	_Done : BOOL;
	_State : DB_COMMAND_EXECUTION_STATE;
	_GetError : BOOL;
	_Logger : Tc3_EventLogger.I_TcMessage;	
	_Connected : BOOL;
	_DataSetLoaded : BOOL;
	_DisconnectingState : DB_COMMAND_DISCONNECTING_STATE;
	_LastException : Exception;
END_VAR

{attribute 'monitoring' := 'call'}
{attribute 'OPC.UA.DA.Property' := '1'}
{attribute 'OPC.UA.DA.Access' := '1'}
PROPERTY Busy : BOOL
GET
Busy := State <> DB_COMMAND_EXECUTION_STATE.IDLING;
END_GET
END_PROPERTY

{attribute 'monitoring' := 'call'}
PROPERTY ClassName : REFERENCE TO STRING
GET
ClassName REF= _ClassName;
END_GET
END_PROPERTY

{attribute 'monitoring' := 'call'}
{attribute 'OPC.UA.DA.Property' := '1'}
{attribute 'OPC.UA.DA.Access' := '1'}
PROPERTY CommandText : REFERENCE TO Tc2_System.T_MaxString
GET
CommandText REF= _ExecutionParameters.CommandText;
END_GET
END_PROPERTY

{attribute 'monitoring' := 'call'}
{attribute 'OPC.UA.DA.Property' := '1'}
{attribute 'OPC.UA.DA.Access' := '1'}
PROPERTY Done : BOOL
GET
Done := _Done;
END_GET
END_PROPERTY

{attribute 'monitoring' := 'call'}
{attribute 'OPC.UA.DA.Property' := '1'}
{attribute 'OPC.UA.DA.Access' := '1'}
PROPERTY Error : BOOL
GET
Error := State = DB_COMMAND_EXECUTION_STATE.IDLING AND_THEN NOT _LastException.Empty;
END_GET
END_PROPERTY

METHOD Execute
VAR
	requestEventTextError : BOOL;	
	requestEventTextErrorCode : HRESULT;
END_VAR
VAR_INST
	errorMessage : STRING(255);	
END_VAR
START:

IF NOT _LastException.Empty THEN
	_GetError := FALSE;
END_IF

IF _GetError THEN
	IF _Logger <> 0 THEN 
		IF _Logger.RequestEventText(
			1033,
			errorMessage,
			SIZEOF(errorMessage),
			bError => requestEventTextError,
			hrErrorCode => requestEventTextErrorCode
		) THEN
			IF requestEventTextError THEN					
				errorMessage := String.Concat2('_Logger.RequestEventText() call error. Error code is ', TO_STRING(requestEventTextErrorCode));
			END_IF
		ELSE
			RETURN;
		END_IF			
	ELSE
		errorMessage :=  'Logger is not specified';
	END_IF				
	
	_LastExceptionHelper.Throw(
		0,
		TO_WSTRING(errorMessage),
		__POUNAME(),
		ClassName,
		CurrentNamespace.Name,
		__POSITION(
	)
	);
	JMP START;	
END_IF

CASE State OF
	DB_COMMAND_EXECUTION_STATE.STARTING:
		MEMSET(destAddr := _ExecutionParameters.TargetBuffer, fillByte := 0, n := _ExecutionParameters.TargetBufferSize);	
		_State := DB_COMMAND_EXECUTION_STATE.CONNECTING;		
		JMP START;		
	
	DB_COMMAND_EXECUTION_STATE.CONNECTING:
		IF _DbConnection.Connect(hDBID := _ExecutionParameters.DBID) THEN
			IF _DbConnection.bError THEN
				_GetError := TRUE;
				_Logger := _DbConnection.ipTcResult;
				_State := DB_COMMAND_EXECUTION_STATE.DISCONNECTING;				
			ELSE
				_Connected := TRUE;
				_State := DB_COMMAND_EXECUTION_STATE.PREPARING;
			END_IF
			
			JMP START;
		END_IF
	
	DB_COMMAND_EXECUTION_STATE.PREPARING:
		IF _DbConnection.CreateCmd(ADR(_Command)) THEN
			IF _DbConnection.bError THEN
				_GetError := TRUE;
				_Logger := _DbConnection.ipTcResult;
				_State := DB_COMMAND_EXECUTION_STATE.DISCONNECTING;				
			ELSE
				_State := DB_COMMAND_EXECUTION_STATE.EXECUTING;
			END_IF
			
			JMP START;
		END_IF
	
	DB_COMMAND_EXECUTION_STATE.EXECUTING:
		IF _ExecutionParameters.MaxRecordsToReadAtTime = 0 THEN
			IF _Command.Execute(ADR(_ExecutionParameters.CommandText), SIZEOF(_ExecutionParameters.CommandText)) THEN
				IF _Command.bError THEN
					_GetError := TRUE;
					_Logger := _Command.ipTcResult;
				END_IF
				
				_State := DB_COMMAND_EXECUTION_STATE.DISCONNECTING;
				
				JMP START;			
			END_IF
		ELSE
			IF _Command.ExecuteDataReturn(ADR(_ExecutionParameters.CommandText), SIZEOF(_ExecutionParameters.CommandText), ADR(_SQLResult)) THEN
				IF _Command.bError THEN
					_GetError := TRUE;
					_Logger := _Command.ipTcResult;
					_State := DB_COMMAND_EXECUTION_STATE.DISCONNECTING;
				ELSE
					_State := DB_COMMAND_EXECUTION_STATE.LOADING_RESULT_DATA_SET;
				END_IF
				
				JMP START;			
			END_IF
		END_IF
		
	DB_COMMAND_EXECUTION_STATE.LOADING_RESULT_DATA_SET:
		IF _SQLResult.Read(
			0,
			_ExecutionParameters.MaxRecordsToReadAtTime,
			_ExecutionParameters.TargetBuffer,
			_ExecutionParameters.TargetBufferSize,
			TRUE,
			TRUE
		) THEN
			IF _SQLResult.bError THEN
				_GetError := TRUE;
				_SQLResult.Release();
				_Logger := _SQLResult.ipTcResult;
			ELSE
				_DataSetLoaded := TRUE;
			END_IF

			_State := DB_COMMAND_EXECUTION_STATE.DISCONNECTING;
			
			JMP START;			
		END_IF

	DB_COMMAND_EXECUTION_STATE.DISCONNECTING:
		CASE _DisconnectingState OF
			DB_COMMAND_DISCONNECTING_STATE.IDLING:
				IF _DataSetLoaded THEN
					_DisconnectingState := DB_COMMAND_DISCONNECTING_STATE.DATA_SET_RELEASING;
				ELSIF _Connected THEN
					_DisconnectingState := DB_COMMAND_DISCONNECTING_STATE.DISCONNECTING;					
				ELSE
					_State := DB_COMMAND_EXECUTION_STATE.IDLING;	
					_Done := _LastException.Empty;	
				END_IF
				
				JMP START;
				
			DB_COMMAND_DISCONNECTING_STATE.DATA_SET_RELEASING:
				IF _SQLResult.Release() THEN
					_DataSetLoaded := FALSE;
					_DisconnectingState := DB_COMMAND_DISCONNECTING_STATE.DISCONNECTING;
					JMP START;										
				END_IF
				
			DB_COMMAND_DISCONNECTING_STATE.DISCONNECTING:
				IF _DbConnection.Disconnect() THEN
					_Connected := FALSE;
					_DisconnectingState := DB_COMMAND_DISCONNECTING_STATE.IDLING;
					JMP START;										
				END_IF
		END_CASE	
END_CASE
END_METHOD

{attribute 'monitoring' := 'call'}
{attribute 'OPC.UA.DA.Property' := '1'}
{attribute 'OPC.UA.DA.Access' := '1'}
PROPERTY LastException : REFERENCE TO Exception
GET
LastException REF= _LastException;
END_GET
END_PROPERTY

METHOD Reset
VAR_OUTPUT
	exception : Exception;
END_VAR
IF Busy THEN
	_LastExceptionHelper.Throw(
		0,
		"Previous command execution is not finished",
		__POUNAME(),
		ClassName,
		CurrentNamespace.Name,
		__POSITION(
	)
	); 
	RETURN;
END_IF

_Done := FALSE;
_State := DB_COMMAND_EXECUTION_STATE.STARTING;
_GetError := FALSE;
_Logger := 0;	
_Connected := FALSE;
_DataSetLoaded := FALSE;
_DisconnectingState := DB_COMMAND_DISCONNECTING_STATE.IDLING;
_LastException.Clear();
END_METHOD

METHOD Start 
VAR_INPUT
	dbId : UDINT;
	commandText : Tc2_System.T_MaxString;
	targetBuffer : PVOID;
	targetBufferSize : UDINT;
	maxRecordsToReadAtTime : UINT;
END_VAR
VAR_OUTPUT
	exception : Exception;
END_VAR
VAR
	executionParameters : POINTER TO DB_COMMAND_EXECUTION_PARAMETERS;
END_VAR
IF Busy THEN
	_LastExceptionHelper.Throw(
		0,
		"Previous command execution is not finished",
		__POUNAME(),
		ClassName,
		CurrentNamespace.Name,
		__POSITION(
	)
	); 
	RETURN;
END_IF

IF maxRecordsToReadAtTime > 0 AND_THEN (targetBuffer = 0 OR_ELSE targetBufferSize = 0) THEN
	_LastExceptionHelper.Throw(
		0,
		"Parameter 'maxRecordsToReadAtTime' is greater then zero, but 'targetBuffer' or 'targetBufferSize' has incorrect values",
		__POUNAME(),
		ClassName,
		CurrentNamespace.Name,
		__POSITION(
	)
	);
	RETURN;
END_IF

_ExecutionParameters.DbId := dbId;
_ExecutionParameters.CommandText := commandText;
_ExecutionParameters.TargetBuffer := targetBuffer; 
_ExecutionParameters.TargetBufferSize := targetBufferSize;
_ExecutionParameters.MaxRecordsToReadAtTime := maxRecordsToReadAtTime;

Reset();
END_METHOD

{attribute 'monitoring' := 'call'}
{attribute 'OPC.UA.DA.Property' := '1'}
{attribute 'OPC.UA.DA.Access' := '1'}
PROPERTY State : DB_COMMAND_EXECUTION_STATE
GET
State := _State;
END_GET
END_PROPERTY

{attribute 'monitoring' := 'call'}
{attribute 'OPC.UA.DA.Property' := '1'}
{attribute 'OPC.UA.DA.Access' := '1'}
PROPERTY Timeout : TIME
GET
Timeout := _Command.tTimeout;
END_GET
SET
_Command.tTimeout := Timeout;
_SQLResult.tTimeout := Timeout;
END_SET
END_PROPERTY

END_FUNCTION_BLOCK

// ---- Database/StoredProcedure/DbProcedureExecutor.TcPOU
{attribute 'no_explicit_call' := 'do not call this function block directly'}
FUNCTION_BLOCK DbProcedureExecutor EXTENDS TC.ToolkitObject IMPLEMENTS TC.IAction
VAR_STAT
	//! <summary>Class name shared by all instances of this function block.</summary>
	_ClassName : STRING := __POUNAME();
END_VAR
VAR	
	_DbConnection : Tc3_Database.FB_SQLDatabaseEvt(sNetID := '', tTimeout := T#10S);	

	_ExecutionParameters : DB_ROCEDURE_EXECUTION_PARAMETERS;

	_StoredProcedure : Tc3_Database.FB_SQLStoredProcedureEvt(sNetID:='', tTimeout := T#10S);
	_SQLResult: Tc3_Database.FB_SQLResultEvt(sNetID := '', tTimeout := T#10S);
	
	_Done : BOOL;
	_State : DB_PROCEDURE_EXECUTION_STATE;
	_GetError : BOOL;
	_Logger : Tc3_EventLogger.I_TcMessage;	
	_Connected : BOOL;
	_Prepared : BOOL;
	_DataSetLoaded : BOOL;
	_DisconnectingState : DB_PROCEDURE_DISCONNECTING_STATE;
	_LastException : Exception;
END_VAR

{attribute 'monitoring' := 'call'}
{attribute 'OPC.UA.DA.Property' := '1'}
{attribute 'OPC.UA.DA.Access' := '1'}
PROPERTY Busy : BOOL
GET
Busy := State <> DB_PROCEDURE_EXECUTION_STATE.IDLING;
END_GET
END_PROPERTY

{attribute 'monitoring' := 'call'}
PROPERTY ClassName : REFERENCE TO STRING
GET
ClassName REF= _ClassName;
END_GET
END_PROPERTY

{attribute 'monitoring' := 'call'}
{attribute 'OPC.UA.DA.Property' := '1'}
{attribute 'OPC.UA.DA.Access' := '1'}
PROPERTY Done : BOOL
GET
Done := _Done;
END_GET
END_PROPERTY

{attribute 'monitoring' := 'call'}
{attribute 'OPC.UA.DA.Property' := '1'}
{attribute 'OPC.UA.DA.Access' := '1'}
PROPERTY Error : BOOL
GET
Error := State = DB_PROCEDURE_EXECUTION_STATE.IDLING AND_THEN NOT _LastException.Empty;
END_GET
END_PROPERTY

METHOD Execute
VAR
	requestEventTextError : BOOL;
	requestEventTextErrorCode : HRESULT;
END_VAR
VAR_INST
	errorMessage : STRING(255);	
END_VAR
START:

IF NOT _LastException.Empty THEN
	_GetError := FALSE;
END_IF

IF _GetError THEN
	IF _Logger <> 0 THEN 
		IF _Logger.RequestEventText(
			1033,
			errorMessage,
			SIZEOF(errorMessage),
			bError => requestEventTextError,
			hrErrorCode => requestEventTextErrorCode
		) THEN
			IF requestEventTextError THEN					
				errorMessage := String.Concat2('_Logger.RequestEventText() call error. Error code is ', TO_STRING(requestEventTextErrorCode));
			END_IF
		ELSE
			RETURN;
		END_IF			
	ELSE
		errorMessage :=  'Logger is not specified';
	END_IF				
	
	_LastExceptionHelper.Throw(
		0,
		TO_WSTRING(errorMessage),
		__POUNAME(),
		ClassName,
		CurrentNamespace.Name,
		__POSITION(
	)
	);
	JMP START;	
END_IF

CASE State OF
	DB_PROCEDURE_EXECUTION_STATE.STARTING:
		MEMSET(destAddr := _ExecutionParameters.TargetBuffer, fillByte := 0, n := _ExecutionParameters.TargetBufferSize);	
		_State := DB_PROCEDURE_EXECUTION_STATE.CONNECTING;			
		JMP START;
				
	DB_PROCEDURE_EXECUTION_STATE.CONNECTING:
		IF _DbConnection.Connect(hDBID := _ExecutionParameters.DBID) THEN
			IF _DbConnection.bError THEN
				_GetError := TRUE;
				_Logger := _DbConnection.ipTcResult;
				_State := DB_PROCEDURE_EXECUTION_STATE.DISCONNECTING;				
			ELSE
				_Connected := TRUE;
				_State := DB_PROCEDURE_EXECUTION_STATE.PREPARING;
			END_IF			

			JMP START;
		END_IF
	
	DB_PROCEDURE_EXECUTION_STATE.PREPARING:
		IF _DbConnection.CreateSP(
			sProcedureName := _ExecutionParameters.ProcedureName,
			pParameterInfo := _ExecutionParameters.ParameterDescriptors,
			cbParameterInfo := _ExecutionParameters.ParameterDescriptorsSize,
			pSQLProcedure := ADR(_StoredProcedure)
		) THEN
			IF _DbConnection.bError THEN
				_GetError := TRUE;
				_Logger := _DbConnection.ipTcResult;
				_State := DB_PROCEDURE_EXECUTION_STATE.DISCONNECTING;				
			ELSE
				_Prepared := TRUE;
				_State := DB_PROCEDURE_EXECUTION_STATE.EXECUTING;
			END_IF
			
			JMP START;
		END_IF
	
	DB_PROCEDURE_EXECUTION_STATE.EXECUTING:
		IF _ExecutionParameters.MaxRecordsToReadAtTime = 0 THEN
			IF _StoredProcedure.Execute(_ExecutionParameters.ParameterValues, _ExecutionParameters.ParameterValuesSize) THEN
				IF _StoredProcedure.bError THEN
					_GetError := TRUE;
					_Logger := _StoredProcedure.ipTcResult;
				END_IF
				
				_State := DB_PROCEDURE_EXECUTION_STATE.DISCONNECTING;
				
				JMP START;			
			END_IF
		ELSE
			IF _StoredProcedure.ExecuteDataReturn(
				_ExecutionParameters.ParameterValues,
				_ExecutionParameters.ParameterValuesSize,
				ADR(_SQLResult)
			) THEN
				IF _StoredProcedure.bError THEN
					_GetError := TRUE;
					_Logger := _StoredProcedure.ipTcResult;
					_State := DB_PROCEDURE_EXECUTION_STATE.DISCONNECTING;
				ELSE
					_State := DB_PROCEDURE_EXECUTION_STATE.LOADING_RESULT_DATA_SET;
				END_IF
								
				JMP START;			
			END_IF
		END_IF
		
	DB_PROCEDURE_EXECUTION_STATE.LOADING_RESULT_DATA_SET:
		IF _SQLResult.Read(
			0,
			_ExecutionParameters.MaxRecordsToReadAtTime,
			_ExecutionParameters.TargetBuffer,
			_ExecutionParameters.TargetBufferSize,
			TRUE,
			TRUE
		) THEN
			IF _SQLResult.bError THEN
				_GetError := TRUE;
				_SQLResult.Release();
				_Logger := _SQLResult.ipTcResult;
			ELSE				
				_DataSetLoaded := TRUE;
			END_IF
			
			_State := DB_PROCEDURE_EXECUTION_STATE.DISCONNECTING;
			
			JMP START;			
		END_IF		

	DB_PROCEDURE_EXECUTION_STATE.DISCONNECTING:
		CASE _DisconnectingState OF
			DB_PROCEDURE_DISCONNECTING_STATE.IDLING:				
				IF _DataSetLoaded THEN
					_DisconnectingState := DB_PROCEDURE_DISCONNECTING_STATE.DATA_SET_RELEASING;
				ELSIF _Prepared THEN
					_DisconnectingState := DB_PROCEDURE_DISCONNECTING_STATE.PARAMETERS_RELEASING;					
				ELSIF _Connected THEN
					_DisconnectingState := DB_PROCEDURE_DISCONNECTING_STATE.DISCONNECTING;					
				ELSE
					_State := DB_PROCEDURE_EXECUTION_STATE.IDLING;				
					_Done := _LastException.Empty;	
				END_IF
				
				JMP START;
				
			DB_PROCEDURE_DISCONNECTING_STATE.DATA_SET_RELEASING:
				IF _SQLResult.Release() THEN
					_DataSetLoaded := FALSE;
					_DisconnectingState := DB_PROCEDURE_DISCONNECTING_STATE.PARAMETERS_RELEASING;
					JMP START;					
				END_IF
			
			DB_PROCEDURE_DISCONNECTING_STATE.PARAMETERS_RELEASING:
				IF _StoredProcedure.Release() THEN
					_Prepared := FALSE;
					_DisconnectingState := DB_PROCEDURE_DISCONNECTING_STATE.DISCONNECTING;
					JMP START;										
				END_IF
				
			DB_PROCEDURE_DISCONNECTING_STATE.DISCONNECTING:
				IF _DbConnection.Disconnect() THEN
					_Connected := FALSE;
					_DisconnectingState := DB_PROCEDURE_DISCONNECTING_STATE.IDLING;
					JMP START;										
				END_IF
		END_CASE	
END_CASE
END_METHOD

{attribute 'monitoring' := 'call'}
{attribute 'OPC.UA.DA.Property' := '1'}
{attribute 'OPC.UA.DA.Access' := '1'}
PROPERTY LastException : REFERENCE TO Exception
GET
LastException REF= _LastException;
END_GET
END_PROPERTY

{attribute 'OPC.UA.DA.Property' := '1'}
{attribute 'OPC.UA.DA.Access' := '1'}
{attribute 'monitoring' := 'call'}
PROPERTY ProcedureName : REFERENCE TO Tc2_System.T_MaxString
GET
ProcedureName REF= _ExecutionParameters.ProcedureName;
END_GET
END_PROPERTY

METHOD Reset 
VAR_OUTPUT
	exception : Exception;
END_VAR
IF Busy THEN
	_LastExceptionHelper.Throw(
		0,
		"Previous command execution is not finished",
		__POUNAME(),
		ClassName,
		CurrentNamespace.Name,
		__POSITION(
	)
	); 
	RETURN;
END_IF

_Done := FALSE;
_State := DB_PROCEDURE_EXECUTION_STATE.STARTING;
_GetError := FALSE;
_Logger := 0;	
_Connected := FALSE;
_Prepared := FALSE;
_DataSetLoaded := FALSE;
_DisconnectingState := DB_PROCEDURE_DISCONNECTING_STATE.IDLING;
_LastException.Clear();
END_METHOD

METHOD Start 
VAR_INPUT
	dbId : UDINT;
	procedureName : Tc2_System.T_MaxString;
	parameterDescriptors : POINTER TO Tc3_Database.ST_SQLSPParameter;
	parameterDescriptorsSize : UDINT;
	parameterValues : PVOID;
	parameterValuesSize : UDINT;
	targetBuffer : PVOID;
	targetBufferSize : UDINT;
	maxRecordsToReadAtTime : UINT;
END_VAR
VAR_OUTPUT
	exception : Exception;
END_VAR
IF Busy THEN
	_LastExceptionHelper.Throw(
		0,
		"Previous command execution is not finished",
		__POUNAME(),
		ClassName,
		CurrentNamespace.Name,
		__POSITION(
	)
	); 
	RETURN;
END_IF

IF maxRecordsToReadAtTime > 0 AND_THEN (targetBuffer = 0 OR_ELSE targetBufferSize = 0) THEN
	_LastExceptionHelper.Throw(
		0,
		"Parameter 'maxRecordsToReadAtTime' is greater then zero, but 'targetBuffer' or 'targetBufferSize' has incorrect values",
		__POUNAME(),
		ClassName,
		CurrentNamespace.Name,
		__POSITION(
	)
	);
	RETURN;
END_IF

_ExecutionParameters.DbId := dbId;
_ExecutionParameters.ProcedureName := procedureName;
_ExecutionParameters.ParameterDescriptors := parameterDescriptors;
_ExecutionParameters.ParameterDescriptorsSize := parameterDescriptorsSize;
_ExecutionParameters.ParameterValues := parameterValues;
_ExecutionParameters.ParameterValuesSize := parameterValuesSize;
_ExecutionParameters.TargetBuffer := targetBuffer; 
_ExecutionParameters.TargetBufferSize := targetBufferSize;
_ExecutionParameters.MaxRecordsToReadAtTime := maxRecordsToReadAtTime;

Reset();
END_METHOD

{attribute 'monitoring' := 'call'}
{attribute 'OPC.UA.DA.Property' := '1'}
{attribute 'OPC.UA.DA.Access' := '1'}
PROPERTY State : DB_PROCEDURE_EXECUTION_STATE
GET
State := _State;
END_GET
END_PROPERTY

{attribute 'monitoring' := 'call'}
{attribute 'OPC.UA.DA.Property' := '1'}
{attribute 'OPC.UA.DA.Access' := '1'}
PROPERTY Timeout : TIME
GET
Timeout := _StoredProcedure.tTimeout;
END_GET
SET
_StoredProcedure.tTimeout := Timeout;
_SQLResult.tTimeout := Timeout;
END_SET
END_PROPERTY

END_FUNCTION_BLOCK

// ---- StateMachine/Finite/FiniteStateMachine.TcPOU
{attribute 'no_explicit_call' := 'do not call this function block directly'}
FUNCTION_BLOCK ABSTRACT FiniteStateMachine EXTENDS ToolkitObject
VAR_INPUT
	{attribute 'OPC.UA.DA' := '0'}
	RequestedCause : STRING;	

	{attribute 'OPC.UA.DA.Access' := '1'}
	CurrentState : REFERENCE TO ProgramState;
	
	{attribute 'OPC.UA.DA.Access' := '1'}
	LastTransition : REFERENCE TO ProgramTransition;
END_VAR
VAR	
	{attribute 'OPC.UA.DA' := '0'}
	_AvailableStates : ARRAY [0..ProgramConstants.MaxStateCount - 1] OF POINTER TO ProgramState;

	{attribute 'OPC.UA.DA' := '0'}
	_AvailableTransitions : ARRAY [0..ProgramConstants.MaxTransitionCount - 1] OF POINTER TO ProgramTransition;
END_VAR

{attribute 'monitoring' := 'call'}
{attribute 'OPC.UA.DA.Property' := '1'}
{attribute 'OPC.UA.DA.Access' := '1'}
PROPERTY ABSTRACT AvailableStateCount : INT(0..ProgramConstants.MaxStateCount - 1)
GET
END_GET
END_PROPERTY

{attribute 'monitoring' := 'call'}
{attribute 'OPC.UA.DA.Property' := '1'}
{attribute 'OPC.UA.DA.Access' := '1'}
PROPERTY ABSTRACT AvailableTransitionCount : INT(0..ProgramConstants.MaxTransitionCount - 1)
GET
END_GET
END_PROPERTY

METHOD INTERNAL Clear
CurrentState REF= 0;
LastTransition REF= 0;

LastException.Clear();
END_METHOD

{attribute 'monitoring' := 'call'}
PROPERTY CurrentStateName : STRING
GET
IF __ISVALIDREF(CurrentState) THEN
	CurrentStateName := CurrentState.Name;
END_IF
END_GET
END_PROPERTY

METHOD Execute
VAR
	newState : POINTER TO ProgramState;
	newTransition : POINTER TO ProgramTransition;
END_VAR
(*IF InTransition THEN
	LastTransition.Execute();
		
	IF LastTransition.Error THEN
		LastException := LastTransition.LastException;
		exceptionSet.AddExisting(LastException);
		RETURN;
	ELSIF LastTransition.Busy THEN
		Execute := TRUE;
		RETURN;
	ELSIF LastTransition.Done THEN
		IF newState := GetStateByName(LastTransition.ToState) THEN
			CurrentState REF= newState^;			
			CurrentState.Enable();
			
			IF CurrentState.Error THEN				
				LastException := CurrentState.LastException;
				exceptionSet.AddExisting(LastException);
				RETURN;
			END_IF
		ELSE
			exceptionSet.AddExisting(LastException);
			RETURN;
		END_IF
	ELSE
		// exceptionFactory.ThrowException(__POSITION(), 0, WString.Concat3("CurrentTransition
		// ", TO_WSTRING(LastTransition.Name), " is not in busy, done or error state"));
		exceptionSet.AddExisting(LastException);
		RETURN;		
	END_IF
END_IF

IF NOT __ISVALIDREF(CurrentState) THEN
	Last//exceptionFactory.ThrowException(__POSITION(), 0, "CurrentState is null");
	exceptionSet.AddExisting(LastException);
	RETURN;
END_IF

IF RequestedCause <> '' THEN
	IF FindTransitionByCause(RequestedCause, transition => newTransition, exception => LastException) THEN
		RequestedCause := '';
		
		IF CurrentState.Busy THEN
			CurrentState.Disable();			
		END_IF
		
		LastTransition REF= newTransition^;
		LastTransition.Start();

		IF NOT LastTransition.Error THEN
			Execute := TRUE;
		ELSE				
			LastException := LastTransition.LastException;
			exceptionSet.AddExisting(LastException);
		END_IF
		
		RETURN;		
	ELSE
		RequestedCause := '';
		exceptionSet.AddExisting(LastException);
		RETURN;
	END_IF
END_IF

IF CurrentState.Busy THEN 
	CurrentState.Execute();
	
	IF CurrentState.Error THEN
		LastException := CurrentState.LastException;
		exceptionSet.AddExisting(LastException);
		RETURN;
	ELSIF NOT CurrentState.Busy THEN
		// exceptionFactory.ThrowException(__POSITION(), 0, WString.Concat3("CurrentState
		// ", TO_WSTRING(CurrentState.Name), " is not in busy or error state"));
		exceptionSet.AddExisting(LastException);
		RETURN;		
	END_IF
END_IF

Execute := TRUE;*)
END_METHOD

METHOD PROTECTED FINAL FindTransitionByCause : POINTER TO ProgramTransition
VAR_INPUT
	cause : STRING;
END_VAR
VAR
	i : INT;
END_VAR
IF NOT __ISVALIDREF(CurrentState) THEN
	// exceptionFactory.ThrowException(__POSITION(), WString.Concat4("Unsupported cause ", TO_WSTRING(cause),
	// " to make transition from state ", TO_WSTRING(CurrentState.Name)));
END_IF

FOR i := 0 TO AvailableTransitionCount - 1 DO
	IF _AvailableTransitions[i]^.FromState = CurrentState.Name AND_THEN _AvailableTransitions[i]^.Cause = cause THEN
		FindTransitionByCause := _AvailableTransitions[i];
		RETURN;
	END_IF
END_FOR

// exceptionFactory.ThrowException(__POSITION(), WString.Concat4("Unsupported cause ", TO_WSTRING(cause),
// " to make transition from state ", TO_WSTRING(CurrentState.Name)));
END_METHOD

METHOD PROTECTED FINAL GetStateByName : POINTER TO ProgramState
VAR_INPUT
	name : STRING;
END_VAR
VAR
	i : INT;
END_VAR
FOR i := 0 TO AvailableStateCount - 1 DO
	IF _AvailableStates[i]^.Name = name THEN
		GetStateByName := _AvailableStates[i];
		RETURN;
	END_IF
END_FOR

//exceptionFactory.ThrowException(__POSITION(), WString.Concat2("Unknown state with name ", TO_WSTRING(name)));
END_METHOD

METHOD Initialize 
VAR
	i, j : INT;
	defaultState : POINTER TO ProgramState;
END_VAR
InternalInitialize(states => _AvailableStates, transitions => _AvailableTransitions, defaultState => defaultState);

IF AvailableStateCount <= 0 OR_ELSE AvailableStateCount > ProgramConstants.MaxStateCount - 1 THEN
	//exceptionFactory.ThrowException(__POSITION(), WString.Concat2("Invalid state count  ", TO_WSTRING(AvailableStateCount)));
END_IF

IF AvailableTransitionCount <= 0 OR_ELSE AvailableTransitionCount > ProgramConstants.MaxTransitionCount - 1 THEN
	//exceptionFactory.ThrowException(__POSITION(), WString.Concat2("Invalid transition count  ", TO_WSTRING(AvailableTransitionCount)));
END_IF

IF defaultState = 0 THEN
	//exceptionFactory.ThrowException(__POSITION(), "Default state is not specified");
END_IF

FOR i := 0 TO AvailableStateCount - 1 DO
	FOR j := 0 TO AvailableTransitionCount - 1 DO
		IF _AvailableStates[i]^.Name = _AvailableTransitions[j]^.FromState
			OR_ELSE _AvailableStates[i]^.Name = _AvailableTransitions[j]^.ToState
		THEN
			_AvailableStates[i]^.RegisterTransition(_AvailableTransitions[j]^);
		END_IF
	END_FOR	
END_FOR

CurrentState REF= defaultState^;
END_METHOD

METHOD PROTECTED ABSTRACT InternalInitialize 
VAR_OUTPUT
	states : ARRAY [0..ProgramConstants.MaxStateCount - 1] OF POINTER TO ProgramState;
	transitions : ARRAY [0..ProgramConstants.MaxTransitionCount - 1] OF POINTER TO ProgramTransition;
	defaultState : POINTER TO ProgramState;
END_VAR
END_METHOD

{attribute 'monitoring' := 'call'}
{attribute 'OPC.UA.DA.Property' := '1'}
{attribute 'OPC.UA.DA.Access' := '1'}
PROPERTY InTransition : BOOL
GET
InTransition := __ISVALIDREF(LastTransition) AND_THEN LastTransition.Busy;
END_GET
END_PROPERTY

{attribute 'monitoring' := 'call'}
PROPERTY LastTransitionName : STRING
GET
IF __ISVALIDREF(LastTransition) THEN
	LastTransitionName := LastTransition.Name;
END_IF
END_GET
END_PROPERTY

END_FUNCTION_BLOCK

// ---- StateMachine/Finite/ProgramState.TcPOU
{attribute 'no_explicit_call' := 'do not call this function block directly'}
FUNCTION_BLOCK ABSTRACT ProgramState EXTENDS ToolkitObject
VAR_OUTPUT
	{attribute 'OPC.UA.DA.Access' := '1'}
	FromTransitions : ARRAY [0..ProgramConstants.MaxTransitionCount - 1] OF STRING;
	{attribute 'OPC.UA.DA.Access' := '1'}
	FromTransitionCount : INT(0..ProgramConstants.MaxTransitionCount - 1);
	{attribute 'OPC.UA.DA.Access' := '1'}
	ToTransitions : ARRAY [0..ProgramConstants.MaxTransitionCount - 1] OF STRING;
	{attribute 'OPC.UA.DA.Access' := '1'}
	ToTransitionCount : INT(0..ProgramConstants.MaxTransitionCount - 1);
END_VAR
VAR
	{attribute 'OPC.UA.DA' := '0'}
	_Busy : BOOL;
	{attribute 'OPC.UA.DA' := '0'}
	_Error : BOOL;

	{attribute 'OPC.UA.DA' := '0'}
	_StateMachine : REFERENCE TO FiniteStateMachine;
END_VAR

{attribute 'monitoring' := 'call'}
{attribute 'OPC.UA.DA.Property' := '1'}
{attribute 'OPC.UA.DA.Access' := '1'}
PROPERTY Busy : BOOL
GET
Busy := _Busy;
END_GET
END_PROPERTY

METHOD Disable
IF _Busy THEN
	_Busy := FALSE;
END_IF
END_METHOD

METHOD Enable
_Busy := TRUE;
_Error := FALSE;
END_METHOD

{attribute 'monitoring' := 'call'}
{attribute 'OPC.UA.DA.Property' := '1'}
{attribute 'OPC.UA.DA.Access' := '1'}
PROPERTY Error : BOOL
GET
Error := _Error;
END_GET
END_PROPERTY

METHOD Execute
END_METHOD

METHOD Initialize 
VAR_INPUT
	stateMachine : REFERENCE TO FiniteStateMachine;
END_VAR
IF NOT __ISVALIDREF(_StateMachine) THEN
	//exceptionFactory.ThrowException(__POSITION(), "programStateMachine is NULL");
END_IF

_StateMachine REF= stateMachine;
END_METHOD

{attribute 'monitoring' := 'call'}
{attribute 'OPC.UA.DA.Property' := '1'}
{attribute 'OPC.UA.DA.Access' := '1'}
PROPERTY Initialized : BOOL
GET
Initialized := __ISVALIDREF(_StateMachine);
END_GET
END_PROPERTY

{attribute 'monitoring' := 'call'}
PROPERTY LastException : REFERENCE TO Exception
GET
LastException REF= _LastException;
END_GET
END_PROPERTY

{attribute 'monitoring' := 'call'}
{attribute 'OPC.UA.DA.Property' := '1'}
{attribute 'OPC.UA.DA.Access' := '1'}
PROPERTY ABSTRACT Name : STRING
GET
END_GET
END_PROPERTY

METHOD INTERNAL FINAL RegisterTransition
VAR_INPUT
	transition : REFERENCE TO ProgramTransition;
END_VAR
IF transition.FromState = Name THEN
	ToTransitions[ToTransitionCount] := transition.Name;
	ToTransitionCount := ToTransitionCount + 1;
ELSIF transition.ToState = Name THEN
	FromTransitions[FromTransitionCount] := transition.Name;
	FromTransitionCount := FromTransitionCount + 1;
END_IF
END_METHOD

END_FUNCTION_BLOCK

// ---- StateMachine/Finite/ProgramTransition.TcPOU
(*!
<summary>{attribute 'OPC.UA.DA.Access' := '1'}</summary>
*)

{attribute 'no_explicit_call' := 'do not call this function block directly'}
FUNCTION_BLOCK ABSTRACT ProgramTransition EXTENDS ToolkitObject IMPLEMENTS IAction
VAR_OUTPUT
	
	//Timeout : TIME := T#3S;
END_VAR
VAR
	{attribute 'OPC.UA.DA' := '0'}
	_Busy : BOOL;
	{attribute 'OPC.UA.DA' := '0'}
	_Done : BOOL;
	{attribute 'OPC.UA.DA' := '0'}
	_Error : BOOL;
	{attribute 'OPC.UA.DA' := '0'}
	_StateMachine : REFERENCE TO FiniteStateMachine;
END_VAR

{attribute 'monitoring' := 'call'}
{attribute 'OPC.UA.DA.Property' := '1'}
{attribute 'OPC.UA.DA.Access' := '1'}
PROPERTY Busy : BOOL
GET
Busy := _Busy;
END_GET
END_PROPERTY

METHOD Cancel
IF _Busy THEN
	_Busy := FALSE;	
END_IF
END_METHOD

{attribute 'monitoring' := 'call'}
{attribute 'OPC.UA.DA.Property' := '1'}
{attribute 'OPC.UA.DA.Access' := '1'}
PROPERTY ABSTRACT Cause : STRING
GET
END_GET
END_PROPERTY

{attribute 'monitoring' := 'call'}
{attribute 'OPC.UA.DA.Property' := '1'}
{attribute 'OPC.UA.DA.Access' := '1'}
PROPERTY Done : BOOL
GET
Done := _Done;
END_GET
END_PROPERTY

{attribute 'monitoring' := 'call'}
{attribute 'OPC.UA.DA.Property' := '1'}
{attribute 'OPC.UA.DA.Access' := '1'}
PROPERTY Error : BOOL
GET
Error := _Error;
END_GET
END_PROPERTY

METHOD Execute
_Busy := FALSE;
_Done := TRUE;
_Error := FALSE;
END_METHOD

{attribute 'monitoring' := 'call'}
{attribute 'OPC.UA.DA.Property' := '1'}
{attribute 'OPC.UA.DA.Access' := '1'}
PROPERTY ABSTRACT FromState : STRING
GET
END_GET
END_PROPERTY

METHOD Initialize
VAR_INPUT
	stateMachine : REFERENCE TO FiniteStateMachine;
END_VAR
IF NOT __ISVALIDREF(_StateMachine) THEN
	//exceptionFactory.ThrowException(__POSITION(), "programStateMachine is NULL");
END_IF

_StateMachine REF= stateMachine;
END_METHOD

{attribute 'monitoring' := 'call'}
{attribute 'OPC.UA.DA.Property' := '1'}
{attribute 'OPC.UA.DA.Access' := '1'}
PROPERTY Initialized : BOOL
GET
Initialized := __ISVALIDREF(_StateMachine);
END_GET
END_PROPERTY

{attribute 'monitoring' := 'call'}
PROPERTY LastException : REFERENCE TO Exception
GET
LastException REF= _LastException;
END_GET
END_PROPERTY

{attribute 'monitoring' := 'call'}
{attribute 'OPC.UA.DA.Property' := '1'}
{attribute 'OPC.UA.DA.Access' := '1'}
PROPERTY ABSTRACT Name : STRING
GET
END_GET
END_PROPERTY

METHOD Start
_Busy := FALSE;
_Done := TRUE;
_Error := FALSE;
END_METHOD

{attribute 'monitoring' := 'call'}
{attribute 'OPC.UA.DA.Property' := '1'}
{attribute 'OPC.UA.DA.Access' := '1'}
PROPERTY ABSTRACT ToState : STRING
GET
END_GET
END_PROPERTY

END_FUNCTION_BLOCK

// ---- StateMachine/Program/ProgramStateMachine.TcPOU
FUNCTION_BLOCK ABSTRACT ProgramStateMachine EXTENDS FiniteStateMachine
VAR
	{attribute 'OPC.UA.DA' := '0'}
	_HaltedState : REFERENCE TO HaltedProgramState;
	{attribute 'OPC.UA.DA' := '0'}
	_ReadyState : REFERENCE TO ReadyProgramState;
	{attribute 'OPC.UA.DA' := '0'}
	_RunningState : REFERENCE TO RunningProgramState;
	{attribute 'OPC.UA.DA' := '0'}
	_SuspendedState : REFERENCE TO SuspendedProgramState;
	
	{attribute 'OPC.UA.DA' := '0'}
	_HaltedToReady : REFERENCE TO HaltedToReadyProgramTransition;
	{attribute 'OPC.UA.DA' := '0'}
	_ReadyToRunning : REFERENCE TO ReadyToRunningProgramTransition;
	{attribute 'OPC.UA.DA' := '0'}
	_RunningToHalted : REFERENCE TO RunningToHaltedProgramTransition;
	{attribute 'OPC.UA.DA' := '0'}
	_RunningToReady : REFERENCE TO RunningToReadyProgramTransition;
	{attribute 'OPC.UA.DA' := '0'}
	_RunningToSuspended : REFERENCE TO RunningToSuspendedProgramTransition;
	{attribute 'OPC.UA.DA' := '0'}
	_SuspendedToRunning : REFERENCE TO SuspendedToRunningProgramTransition;
	{attribute 'OPC.UA.DA' := '0'}
	_SuspendedToHalted : REFERENCE TO SuspendedToHaltedProgramTransition;
	{attribute 'OPC.UA.DA' := '0'}
	_SuspendedToReady : REFERENCE TO SuspendedToReadyProgramTransition;
	{attribute 'OPC.UA.DA' := '0'}
	_ReadyToHalted : REFERENCE TO ReadyToHaltedProgramTransition;
END_VAR

{attribute 'monitoring' := 'call'}
{attribute 'OPC.UA.DA.Property' := '1'}
{attribute 'OPC.UA.DA.Access' := '1'}
PROPERTY AvailableStateCount : INT (0..(ProgramConstants.MaxStateCount - 1))
GET
AvailableStateCount := 4;
END_GET
END_PROPERTY

{attribute 'monitoring' := 'call'}
{attribute 'OPC.UA.DA.Property' := '1'}
{attribute 'OPC.UA.DA.Access' := '1'}
PROPERTY AvailableTransitionCount : INT (0..(ProgramConstants.MaxTransitionCount - 1))
GET
AvailableTransitionCount := 9;
END_GET
END_PROPERTY

METHOD PROTECTED ABSTRACT GetStateAndTransitionInstances
VAR_OUTPUT
	haltedState : POINTER TO HaltedProgramState;
	readyState : POINTER TO ReadyProgramState;
	runningState : POINTER TO RunningProgramState;
	suspendedState : POINTER TO SuspendedProgramState;
	
	haltedToReady : POINTER TO HaltedToReadyProgramTransition;
	readyToRunning : POINTER TO ReadyToRunningProgramTransition;
	runningToHalted : POINTER TO RunningToHaltedProgramTransition;
	runningToReady : POINTER TO RunningToReadyProgramTransition;
	runningToSuspended : POINTER TO RunningToSuspendedProgramTransition;
	suspendedToRunning : POINTER TO SuspendedToRunningProgramTransition;
	suspendedToHalted : POINTER TO SuspendedToHaltedProgramTransition;
	suspendedToReady : POINTER TO SuspendedToReadyProgramTransition;
	readyToHalted : POINTER TO ReadyToHaltedProgramTransition;	
END_VAR
END_METHOD

{attribute 'TcRpcEnable':='1'}
METHOD FINAL Halt : BOOL
VAR_OUTPUT
	errorMessage : ERROR_MESSAGE;
END_VAR
__TRY
	FindTransitionByCause(__POUNAME());
	RequestedCause := __POUNAME();
	Halt := TRUE;
__CATCH
	errorMessage := ExceptionHelper.LastException.ToString(FALSE);
	ExceptionHelper.Cleanup();
__ENDTRY
END_METHOD

METHOD PROTECTED InternalInitialize 
VAR_OUTPUT
	states : ARRAY [0..ProgramConstants.MaxStateCount - 1] OF POINTER TO ProgramState;
	transitions : ARRAY [0..ProgramConstants.MaxTransitionCount - 1] OF POINTER TO ProgramTransition;
	defaultState : POINTER TO ProgramState;
END_VAR
VAR
	haltedState : POINTER TO HaltedProgramState;
	readyState : POINTER TO ReadyProgramState;
	runningState : POINTER TO RunningProgramState;
	suspendedState : POINTER TO SuspendedProgramState;
	
	haltedToReady : POINTER TO HaltedToReadyProgramTransition;
	readyToRunning : POINTER TO ReadyToRunningProgramTransition;
	runningToHalted : POINTER TO RunningToHaltedProgramTransition;
	runningToReady : POINTER TO RunningToReadyProgramTransition;
	runningToSuspended : POINTER TO RunningToSuspendedProgramTransition;
	suspendedToRunning : POINTER TO SuspendedToRunningProgramTransition;
	suspendedToHalted : POINTER TO SuspendedToHaltedProgramTransition;
	suspendedToReady : POINTER TO SuspendedToReadyProgramTransition;
	readyToHalted : POINTER TO ReadyToHaltedProgramTransition;	
END_VAR
GetStateAndTransitionInstances(	
	haltedState => haltedState, 
	readyState => readyState, 
	runningState => runningState, 
	suspendedState => suspendedState,
	
	haltedToReady => haltedToReady,
	readyToRunning => readyToRunning,
	runningToHalted => runningToHalted,
	runningToReady => runningToReady,
	runningToSuspended => runningToSuspended,
	suspendedToRunning => suspendedToRunning,
	suspendedToHalted => suspendedToHalted,
	suspendedToReady => suspendedToReady,
	readyToHalted => readyToHalted
);	

_HaltedState REF= haltedState^;
_ReadyState REF= readyState^;
_RunningState REF= runningState^;
_SuspendedState REF= suspendedState^;

_HaltedToReady REF= haltedToReady^;
_ReadyToRunning REF= readyToRunning^;
_RunningToHalted REF= runningToHalted^;
_RunningToReady REF= runningToReady^;
_RunningToSuspended REF= runningToSuspended^;
_SuspendedToRunning REF= suspendedToRunning^;
_SuspendedToHalted REF= suspendedToHalted^;
_SuspendedToReady REF= suspendedToReady^;
_ReadyToHalted REF= readyToHalted^;

states[0] := haltedState;
states[1] := readyState;
states[2] := runningState;
states[3] := suspendedState;

transitions[0] := haltedToReady;
transitions[1] := readyToRunning;
transitions[2] := runningToHalted;
transitions[3] := runningToReady;
transitions[4] := runningToSuspended;
transitions[5] := suspendedToRunning;
transitions[6] := suspendedToHalted;
transitions[7] := suspendedToReady;
transitions[8] := readyToHalted;

defaultState := readyState;
END_METHOD

{attribute 'TcRpcEnable':='1'}
METHOD FINAL Reset : BOOL
VAR_OUTPUT
	errorMessage : ERROR_MESSAGE;
END_VAR
__TRY
	FindTransitionByCause(__POUNAME());
	RequestedCause := __POUNAME();
	Reset := TRUE;
__CATCH
	errorMessage := ExceptionHelper.LastException.ToString(FALSE);
	ExceptionHelper.Cleanup();
__ENDTRY
END_METHOD

{attribute 'TcRpcEnable':='1'}
METHOD FINAL Resume : BOOL
VAR_OUTPUT
	errorMessage : ERROR_MESSAGE;
END_VAR
__TRY
	FindTransitionByCause(__POUNAME());
	RequestedCause := __POUNAME();
	Resume := TRUE;	
__CATCH
	errorMessage := ExceptionHelper.LastException.ToString(FALSE);
	ExceptionHelper.Cleanup();
__ENDTRY
END_METHOD

{attribute 'TcRpcEnable':='1'}
METHOD FINAL Start: BOOL
VAR_OUTPUT
	errorMessage : ERROR_MESSAGE;
END_VAR
__TRY
	FindTransitionByCause(__POUNAME());
	RequestedCause := __POUNAME();
	Start := TRUE;
__CATCH
	errorMessage := ExceptionHelper.LastException.ToString(FALSE);
	ExceptionHelper.Cleanup();
__ENDTRY
END_METHOD

{attribute 'TcRpcEnable':='1'}
METHOD FINAL Suspend : BOOL
VAR_OUTPUT
	errorMessage : ERROR_MESSAGE;
END_VAR
__TRY
	FindTransitionByCause(__POUNAME());
	RequestedCause := __POUNAME();
	Suspend := TRUE;
__CATCH
	errorMessage := ExceptionHelper.LastException.ToString(FALSE);
	ExceptionHelper.Cleanup();
__ENDTRY
END_METHOD

END_FUNCTION_BLOCK

// ---- StateMachine/Program/States/HaltedProgramState.TcPOU
FUNCTION_BLOCK ABSTRACT HaltedProgramState EXTENDS ProgramState

{attribute 'monitoring' := 'call'}
{attribute 'OPC.UA.DA.Property' := '1'}
{attribute 'OPC.UA.DA.Access' := '1'}
PROPERTY FINAL Name : STRING
GET
Name := 'Halted';
END_GET
END_PROPERTY

END_FUNCTION_BLOCK

// ---- StateMachine/Program/States/ReadyProgramState.TcPOU
FUNCTION_BLOCK ABSTRACT ReadyProgramState EXTENDS ProgramState

{attribute 'monitoring' := 'call'}
{attribute 'OPC.UA.DA.Property' := '1'}
{attribute 'OPC.UA.DA.Access' := '1'}
PROPERTY FINAL Name : STRING
GET
Name := 'Ready';
END_GET
END_PROPERTY

END_FUNCTION_BLOCK

// ---- StateMachine/Program/States/RunningProgramState.TcPOU
FUNCTION_BLOCK ABSTRACT RunningProgramState EXTENDS ProgramState

{attribute 'monitoring' := 'call'}
{attribute 'OPC.UA.DA.Property' := '1'}
{attribute 'OPC.UA.DA.Access' := '1'}
PROPERTY FINAL Name : STRING
GET
Name := 'Running';
END_GET
END_PROPERTY

END_FUNCTION_BLOCK

// ---- StateMachine/Program/States/SuspendedProgramState.TcPOU
FUNCTION_BLOCK ABSTRACT SuspendedProgramState EXTENDS ProgramState

{attribute 'monitoring' := 'call'}
{attribute 'OPC.UA.DA.Property' := '1'}
{attribute 'OPC.UA.DA.Access' := '1'}
PROPERTY FINAL Name : STRING
GET
Name := 'Suspended';
END_GET
END_PROPERTY

END_FUNCTION_BLOCK

// ---- StateMachine/Program/Transitions/HaltedToReadyProgramTransition.TcPOU
FUNCTION_BLOCK ABSTRACT HaltedToReadyProgramTransition EXTENDS ProgramTransition

{attribute 'monitoring' := 'call'}
{attribute 'OPC.UA.DA.Property' := '1'}
{attribute 'OPC.UA.DA.Access' := '1'}
PROPERTY FINAL Cause : STRING
GET
Cause := 'Reset';
END_GET
END_PROPERTY

{attribute 'monitoring' := 'call'}
{attribute 'OPC.UA.DA.Property' := '1'}
{attribute 'OPC.UA.DA.Access' := '1'}
PROPERTY FINAL FromState : STRING
GET
FromState := 'Halted';
END_GET
END_PROPERTY

{attribute 'monitoring' := 'call'}
{attribute 'OPC.UA.DA.Property' := '1'}
{attribute 'OPC.UA.DA.Access' := '1'}
PROPERTY FINAL Name : STRING
GET
Name := 'HaltedToReady';
END_GET
END_PROPERTY

{attribute 'monitoring' := 'call'}
{attribute 'OPC.UA.DA.Property' := '1'}
{attribute 'OPC.UA.DA.Access' := '1'}
PROPERTY FINAL ToState : STRING
GET
ToState := 'Ready';
END_GET
END_PROPERTY

END_FUNCTION_BLOCK

// ---- StateMachine/Program/Transitions/ReadyToRunningProgramTransition.TcPOU
FUNCTION_BLOCK ABSTRACT ReadyToRunningProgramTransition EXTENDS ProgramTransition

{attribute 'monitoring' := 'call'}
{attribute 'OPC.UA.DA.Property' := '1'}
{attribute 'OPC.UA.DA.Access' := '1'}
PROPERTY FINAL Cause : STRING
GET
Cause := 'Start';
END_GET
END_PROPERTY

{attribute 'monitoring' := 'call'}
{attribute 'OPC.UA.DA.Property' := '1'}
{attribute 'OPC.UA.DA.Access' := '1'}
PROPERTY FINAL FromState : STRING
GET
FromState := 'Ready';
END_GET
END_PROPERTY

{attribute 'monitoring' := 'call'}
{attribute 'OPC.UA.DA.Property' := '1'}
{attribute 'OPC.UA.DA.Access' := '1'}
PROPERTY FINAL Name : STRING
GET
Name := 'ReadyToRunning';
END_GET
END_PROPERTY

{attribute 'monitoring' := 'call'}
{attribute 'OPC.UA.DA.Property' := '1'}
{attribute 'OPC.UA.DA.Access' := '1'}
PROPERTY FINAL ToState : STRING
GET
ToState := 'Running';
END_GET
END_PROPERTY

END_FUNCTION_BLOCK

// ---- StateMachine/Program/Transitions/RunningToHaltedProgramTransition.TcPOU
FUNCTION_BLOCK ABSTRACT RunningToHaltedProgramTransition EXTENDS ProgramTransition

{attribute 'monitoring' := 'call'}
{attribute 'OPC.UA.DA.Property' := '1'}
{attribute 'OPC.UA.DA.Access' := '1'}
PROPERTY FINAL Cause : STRING
GET
Cause := 'Halt';
END_GET
END_PROPERTY

{attribute 'monitoring' := 'call'}
{attribute 'OPC.UA.DA.Property' := '1'}
{attribute 'OPC.UA.DA.Access' := '1'}
PROPERTY FINAL FromState : STRING
GET
FromState := 'Running';
END_GET
END_PROPERTY

{attribute 'monitoring' := 'call'}
{attribute 'OPC.UA.DA.Property' := '1'}
{attribute 'OPC.UA.DA.Access' := '1'}
PROPERTY FINAL Name : STRING
GET
Name := 'RunningToHalted';
END_GET
END_PROPERTY

{attribute 'monitoring' := 'call'}
{attribute 'OPC.UA.DA.Property' := '1'}
{attribute 'OPC.UA.DA.Access' := '1'}
PROPERTY FINAL ToState : STRING
GET
ToState := 'Halted';
END_GET
END_PROPERTY

END_FUNCTION_BLOCK

// ---- StateMachine/Program/Transitions/RunningToReadyProgramTransition.TcPOU
FUNCTION_BLOCK ABSTRACT RunningToReadyProgramTransition EXTENDS ProgramTransition

{attribute 'monitoring' := 'call'}
{attribute 'OPC.UA.DA.Property' := '1'}
{attribute 'OPC.UA.DA.Access' := '1'}
PROPERTY FINAL Cause : STRING
GET
Cause := '';
END_GET
END_PROPERTY

{attribute 'monitoring' := 'call'}
{attribute 'OPC.UA.DA.Property' := '1'}
{attribute 'OPC.UA.DA.Access' := '1'}
PROPERTY FINAL FromState : STRING
GET
FromState := 'Running';
END_GET
END_PROPERTY

{attribute 'monitoring' := 'call'}
{attribute 'OPC.UA.DA.Property' := '1'}
{attribute 'OPC.UA.DA.Access' := '1'}
PROPERTY FINAL Name : STRING
GET
Name := 'RunningToReady';
END_GET
END_PROPERTY

{attribute 'monitoring' := 'call'}
{attribute 'OPC.UA.DA.Property' := '1'}
{attribute 'OPC.UA.DA.Access' := '1'}
PROPERTY FINAL ToState : STRING
GET
ToState := 'Ready';
END_GET
END_PROPERTY

END_FUNCTION_BLOCK

// ---- StateMachine/Program/Transitions/RunningToSuspendedProgramTransition.TcPOU
FUNCTION_BLOCK ABSTRACT RunningToSuspendedProgramTransition EXTENDS ProgramTransition

{attribute 'monitoring' := 'call'}
{attribute 'OPC.UA.DA.Property' := '1'}
{attribute 'OPC.UA.DA.Access' := '1'}
PROPERTY FINAL Cause : STRING
GET
Cause := 'Suspend';
END_GET
END_PROPERTY

{attribute 'monitoring' := 'call'}
{attribute 'OPC.UA.DA.Property' := '1'}
{attribute 'OPC.UA.DA.Access' := '1'}
PROPERTY FINAL FromState : STRING
GET
FromState := 'Running';
END_GET
END_PROPERTY

{attribute 'monitoring' := 'call'}
{attribute 'OPC.UA.DA.Property' := '1'}
{attribute 'OPC.UA.DA.Access' := '1'}
PROPERTY FINAL Name : STRING
GET
Name := 'RunningToSuspended';
END_GET
END_PROPERTY

{attribute 'monitoring' := 'call'}
{attribute 'OPC.UA.DA.Property' := '1'}
{attribute 'OPC.UA.DA.Access' := '1'}
PROPERTY FINAL ToState : STRING
GET
ToState := 'Suspended';
END_GET
END_PROPERTY

END_FUNCTION_BLOCK

// ---- StateMachine/Program/Transitions/SuspendedToRunningProgramTransition.TcPOU
FUNCTION_BLOCK ABSTRACT SuspendedToRunningProgramTransition EXTENDS ProgramTransition

{attribute 'monitoring' := 'call'}
{attribute 'OPC.UA.DA.Property' := '1'}
{attribute 'OPC.UA.DA.Access' := '1'}
PROPERTY FINAL Cause : STRING
GET
Cause := 'Resume';
END_GET
END_PROPERTY

{attribute 'monitoring' := 'call'}
{attribute 'OPC.UA.DA.Property' := '1'}
{attribute 'OPC.UA.DA.Access' := '1'}
PROPERTY FINAL FromState : STRING
GET
FromState := 'Suspended';
END_GET
END_PROPERTY

{attribute 'monitoring' := 'call'}
{attribute 'OPC.UA.DA.Property' := '1'}
{attribute 'OPC.UA.DA.Access' := '1'}
PROPERTY FINAL Name : STRING
GET
Name := 'SuspendedToRunning';
END_GET
END_PROPERTY

{attribute 'monitoring' := 'call'}
{attribute 'OPC.UA.DA.Property' := '1'}
{attribute 'OPC.UA.DA.Access' := '1'}
PROPERTY FINAL ToState : STRING
GET
ToState := 'Running';
END_GET
END_PROPERTY

END_FUNCTION_BLOCK

// ---- StateMachine/Program/Transitions/SuspendedToHaltedProgramTransition.TcPOU
FUNCTION_BLOCK ABSTRACT SuspendedToHaltedProgramTransition EXTENDS ProgramTransition

{attribute 'monitoring' := 'call'}
{attribute 'OPC.UA.DA.Property' := '1'}
{attribute 'OPC.UA.DA.Access' := '1'}
PROPERTY FINAL Cause : STRING
GET
Cause := 'Halt';
END_GET
END_PROPERTY

{attribute 'monitoring' := 'call'}
{attribute 'OPC.UA.DA.Property' := '1'}
{attribute 'OPC.UA.DA.Access' := '1'}
PROPERTY FINAL FromState : STRING
GET
FromState := 'Suspended';
END_GET
END_PROPERTY

{attribute 'monitoring' := 'call'}
{attribute 'OPC.UA.DA.Property' := '1'}
{attribute 'OPC.UA.DA.Access' := '1'}
PROPERTY FINAL Name : STRING
GET
Name := 'SuspendedToHalted';
END_GET
END_PROPERTY

{attribute 'monitoring' := 'call'}
{attribute 'OPC.UA.DA.Property' := '1'}
{attribute 'OPC.UA.DA.Access' := '1'}
PROPERTY FINAL ToState : STRING
GET
ToState := 'Halted';
END_GET
END_PROPERTY

END_FUNCTION_BLOCK

// ---- StateMachine/Program/Transitions/SuspendedToReadyProgramTransition.TcPOU
FUNCTION_BLOCK ABSTRACT SuspendedToReadyProgramTransition EXTENDS ProgramTransition

{attribute 'monitoring' := 'call'}
{attribute 'OPC.UA.DA.Property' := '1'}
{attribute 'OPC.UA.DA.Access' := '1'}
PROPERTY FINAL Cause : STRING
GET
Cause := 'Reset';
END_GET
END_PROPERTY

{attribute 'monitoring' := 'call'}
{attribute 'OPC.UA.DA.Property' := '1'}
{attribute 'OPC.UA.DA.Access' := '1'}
PROPERTY FINAL FromState : STRING
GET
FromState := 'Suspended';
END_GET
END_PROPERTY

{attribute 'monitoring' := 'call'}
{attribute 'OPC.UA.DA.Property' := '1'}
{attribute 'OPC.UA.DA.Access' := '1'}
PROPERTY FINAL Name : STRING
GET
Name := 'SuspendedToReady';
END_GET
END_PROPERTY

{attribute 'monitoring' := 'call'}
{attribute 'OPC.UA.DA.Property' := '1'}
{attribute 'OPC.UA.DA.Access' := '1'}
PROPERTY FINAL ToState : STRING
GET
ToState := 'Ready';
END_GET
END_PROPERTY

END_FUNCTION_BLOCK

// ---- StateMachine/Program/Transitions/ReadyToHaltedProgramTransition.TcPOU
FUNCTION_BLOCK ABSTRACT ReadyToHaltedProgramTransition EXTENDS ProgramTransition

{attribute 'monitoring' := 'call'}
{attribute 'OPC.UA.DA.Property' := '1'}
{attribute 'OPC.UA.DA.Access' := '1'}
PROPERTY FINAL Cause : STRING
GET
Cause := '';
END_GET
END_PROPERTY

{attribute 'monitoring' := 'call'}
{attribute 'OPC.UA.DA.Property' := '1'}
{attribute 'OPC.UA.DA.Access' := '1'}
PROPERTY FINAL FromState : STRING
GET
FromState := '';
END_GET
END_PROPERTY

{attribute 'monitoring' := 'call'}
{attribute 'OPC.UA.DA.Property' := '1'}
{attribute 'OPC.UA.DA.Access' := '1'}
PROPERTY FINAL Name : STRING
GET
Name := 'ReadyToHalted';
END_GET
END_PROPERTY

{attribute 'monitoring' := 'call'}
{attribute 'OPC.UA.DA.Property' := '1'}
{attribute 'OPC.UA.DA.Access' := '1'}
PROPERTY FINAL ToState : STRING
GET
ToState := 'Halted';
END_GET
END_PROPERTY

END_FUNCTION_BLOCK

// ---- StateMachine/UnifiedProgram/States/HaltedUnifiedProgramState.TcPOU
FUNCTION_BLOCK HaltedUnifiedProgramState EXTENDS HaltedProgramState
VAR_STAT
	//! <summary>Class name shared by all instances of this function block.</summary>
	{attribute 'OPC.UA.DA' := '0'}
	_ClassName : STRING := __POUNAME();
END_VAR

{attribute 'monitoring' := 'call'}
PROPERTY ClassName : REFERENCE TO STRING
GET
ClassName REF= _ClassName;
END_GET
END_PROPERTY

END_FUNCTION_BLOCK

// ---- StateMachine/UnifiedProgram/States/ReadyUnifiedProgramState.TcPOU
FUNCTION_BLOCK ReadyUnifiedProgramState EXTENDS ReadyProgramState
VAR_STAT
	//! <summary>Class name shared by all instances of this function block.</summary>
	{attribute 'OPC.UA.DA' := '0'}
	_ClassName : STRING := __POUNAME();
END_VAR

{attribute 'monitoring' := 'call'}
PROPERTY ClassName : REFERENCE TO STRING
GET
ClassName REF= _ClassName;
END_GET
END_PROPERTY

END_FUNCTION_BLOCK

// ---- StateMachine/UnifiedProgram/States/RunningUnifiedProgramState.TcPOU
FUNCTION_BLOCK RunningUnifiedProgramState EXTENDS RunningProgramState
VAR_STAT
	//! <summary>Class name shared by all instances of this function block.</summary>
	{attribute 'OPC.UA.DA' := '0'}
	_ClassName : STRING := __POUNAME();
END_VAR

{attribute 'monitoring' := 'call'}
PROPERTY ClassName : REFERENCE TO STRING
GET
ClassName REF= _ClassName;
END_GET
END_PROPERTY

END_FUNCTION_BLOCK

// ---- StateMachine/UnifiedProgram/States/SuspendedUnifiedProgramState.TcPOU
FUNCTION_BLOCK SuspendedUnifiedProgramState EXTENDS SuspendedProgramState
VAR_STAT
	//! <summary>Class name shared by all instances of this function block.</summary>
	{attribute 'OPC.UA.DA' := '0'}
	_ClassName : STRING := __POUNAME();
END_VAR

{attribute 'monitoring' := 'call'}
PROPERTY ClassName : REFERENCE TO STRING
GET
ClassName REF= _ClassName;
END_GET
END_PROPERTY

END_FUNCTION_BLOCK

// ---- StateMachine/UnifiedProgram/StepModels/UnifiedProgramExecutedStep.TcPOU
FUNCTION_BLOCK UnifiedProgramExecutedStep EXTENDS ToolkitObject
VAR_OUTPUT
	StepIndex : INT;
	
	Suspend : BOOL;
	Complete : BOOL;
	
	Actions : ARRAY [0..UnifiedProgramConstants.MaxStepActionsCount - 1] OF POINTER TO UnifiedProgramExecutedStepAction;
	ActionCount : INT;
	
	Transitions : ARRAY [0..UnifiedProgramConstants.MaxStepTransitionsCount - 1] OF POINTER TO UnifiedProgramExecutedStepTransition;
	TransitionCount : INT;
END_VAR
VAR_STAT
	//! <summary>Class name shared by all instances of this function block.</summary>
	{attribute 'OPC.UA.DA' := '0'}
	_ClassName : STRING := __POUNAME();
END_VAR

{attribute 'monitoring' := 'call'}
PROPERTY ClassName : REFERENCE TO STRING
GET
ClassName REF= _ClassName;
END_GET
END_PROPERTY

METHOD Clear
VAR
	i : INT;
END_VAR
Suspend := FALSE;
Complete := FALSE;

FOR i := 0 TO UnifiedProgramConstants.MaxStepActionsCount - 1 DO
	IF Actions[i] <> 0 THEN
		__DELETE(Actions[i]);		
	END_IF
END_FOR

ActionCount := 0;

FOR i := 0 TO UnifiedProgramConstants.MaxStepTransitionsCount - 1 DO
	IF Transitions[i] <> 0 THEN
		__DELETE(Actions[i]);		
	END_IF	
END_FOR

TransitionCount := 0;
END_METHOD

METHOD Decode : BOOL
VAR_INPUT
	stepIndex : INT; 
	step : REFERENCE TO UNIFIED_PROGRAM_STEP;
END_VAR
VAR
	i : INT;
END_VAR
StepIndex := stepIndex;	
Suspend := step.Suspend;
Complete := step.Complete;

FOR i := 0 TO UnifiedProgramConstants.MaxStepActionsCount - 1 DO
	IF step.Actions[i].Name <> '' THEN
		Actions[i] := UnifiedProgramExecutedStepHelper.CreateActionInstance(actionName := step.Actions[i].Name, exception => exception);
		
		IF Actions[i] = 0 THEN
			RETURN;
		END_IF
		
		IF NOT Actions[i]^.Decode(actionIndex := i, stepAction := step.Actions[i], exception => exception) THEN
			RETURN;
		END_IF
	ELSE
		EXIT;
	END_IF
END_FOR

(*FOR i := 0 TO UnifiedProgramConstants.MaxStepTransitionsCount - 1 DO
		Transitions[i] := UnifiedProgramExecutedStepHelper.CreateActionInstance(step.Actions[i].Name, exception => exception);
		
		IF Actions[i] = 0 THEN
			RETURN;
		END_IF
		
		IF NOT Actions[i]^.Decode(i, step.Actions[i], exception => exception) THEN
			RETURN;
		END_IF
	ELSE
		EXIT;
	END_IF
END_FOR*)
END_METHOD

END_FUNCTION_BLOCK

// ---- StateMachine/UnifiedProgram/StepModels/UnifiedProgramExecutedStepAction.TcPOU
FUNCTION_BLOCK ABSTRACT UnifiedProgramExecutedStepAction EXTENDS ToolkitObject
VAR_STAT
	//! <summary>Class name shared by all instances of this function block.</summary>
	{attribute 'OPC.UA.DA' := '0'}
	_ClassName : STRING := __POUNAME();
END_VAR

METHOD ABSTRACT Decode : BOOL
VAR_INPUT
	actionIndex : INT; 
	stepAction : REFERENCE TO UNIFIED_PROGRAM_STEP_ACTION;
END_VAR
END_METHOD

END_FUNCTION_BLOCK

// ---- StateMachine/UnifiedProgram/StepModels/UnifiedProgramExecutedStepTransition.TcPOU
FUNCTION_BLOCK UnifiedProgramExecutedStepTransition EXTENDS ToolkitObject
VAR_STAT
	//! <summary>Class name shared by all instances of this function block.</summary>
	{attribute 'OPC.UA.DA' := '0'}
	_ClassName : STRING := __POUNAME();
END_VAR

{attribute 'monitoring' := 'call'}
PROPERTY ClassName : REFERENCE TO STRING
GET
ClassName REF= _ClassName;
END_GET
END_PROPERTY

METHOD Decode : BOOL
VAR_INPUT
	transitionIndex : INT; 
	stepTransition : REFERENCE TO UNIFIED_PROGRAM_STEP_TRANSITION;
END_VAR
END_METHOD

END_FUNCTION_BLOCK

// ---- StateMachine/UnifiedProgram/StepModels/UnifiedProgramExecutedStepHelper.TcPOU
PROGRAM UnifiedProgramExecutedStepHelper

METHOD CreateActionInstance : POINTER TO UnifiedProgramExecutedStepAction
VAR_INPUT
	actionName : STRING;
END_VAR
END_METHOD

METHOD CreateTransitionConditionInstance : POINTER TO UnifiedProgramExecutedStepTransitionCondition
VAR_INPUT
	conditionName : STRING;
END_VAR
END_METHOD

END_PROGRAM

// ---- StateMachine/UnifiedProgram/StepModels/UnifiedProgramExecutedStepTransitionCondition.TcPOU
FUNCTION_BLOCK ABSTRACT UnifiedProgramExecutedStepTransitionCondition EXTENDS ToolkitObject
VAR_STAT
	//! <summary>Class name shared by all instances of this function block.</summary>
	{attribute 'OPC.UA.DA' := '0'}
	_ClassName : STRING := __POUNAME();
END_VAR

METHOD ABSTRACT Decode : BOOL
VAR_INPUT
	transitionIndex : INT; 
	stepTransition : REFERENCE TO UNIFIED_PROGRAM_STEP_TRANSITION;
END_VAR
END_METHOD

END_FUNCTION_BLOCK

// ---- StateMachine/UnifiedProgram/Transitions/HaltedToReadyUnifiedProgramTransition.TcPOU
FUNCTION_BLOCK HaltedToReadyUnifiedProgramTransition EXTENDS HaltedToReadyProgramTransition
VAR_STAT
	//! <summary>Class name shared by all instances of this function block.</summary>
	{attribute 'OPC.UA.DA' := '0'}
	_ClassName : STRING := __POUNAME();
END_VAR

{attribute 'monitoring' := 'call'}
PROPERTY ClassName : REFERENCE TO STRING
GET
ClassName REF= _ClassName;
END_GET
END_PROPERTY

END_FUNCTION_BLOCK

// ---- StateMachine/UnifiedProgram/Transitions/ReadyToHaltedUnifiedProgramTransition.TcPOU
FUNCTION_BLOCK ReadyToHaltedUnifiedProgramTransition EXTENDS ReadyToHaltedProgramTransition
VAR_STAT
	//! <summary>Class name shared by all instances of this function block.</summary>
	{attribute 'OPC.UA.DA' := '0'}
	_ClassName : STRING := __POUNAME();
END_VAR

{attribute 'monitoring' := 'call'}
PROPERTY ClassName : REFERENCE TO STRING
GET
ClassName REF= _ClassName;
END_GET
END_PROPERTY

END_FUNCTION_BLOCK

// ---- StateMachine/UnifiedProgram/Transitions/ReadyToRunningUnifiedProgramTransition.TcPOU
FUNCTION_BLOCK ReadyToRunningUnifiedProgramTransition EXTENDS ReadyToRunningProgramTransition
VAR_STAT
	//! <summary>Class name shared by all instances of this function block.</summary>
	{attribute 'OPC.UA.DA' := '0'}
	_ClassName : STRING := __POUNAME();
END_VAR

{attribute 'monitoring' := 'call'}
PROPERTY ClassName : REFERENCE TO STRING
GET
ClassName REF= _ClassName;
END_GET
END_PROPERTY

METHOD Start
VAR
	i : INT;
	executedSteps : ARRAY [0..UnifiedProgramConstants.MaxStepCount - 1] OF UNIFIED_PROGRAM_EXECUTED_STEP;
	executedStepCount : INT;
END_VAR
UnifiedProgramStateMachine^.LastException.Clear();
UnifiedProgramStateMachine^.StepExecutor.Reset();

FOR i := 0 TO UnifiedProgramConstants.MaxStepCount - 1 DO
	executedSteps[i].StepIndex := i;
	ExecutedSteps[i].Step REF= UnifiedProgramStateMachine^.Configuration.Steps[i];
	
	executedStepCount := executedStepCount + 1;
	
	IF UnifiedProgramStateMachine^.Configuration.Steps[i].Complete THEN
		EXIT;
	END_IF
END_FOR

_Busy := FALSE;
_Done := TRUE;
_Error := FALSE;
END_METHOD

PROPERTY UnifiedProgramStateMachine : POINTER TO UnifiedProgramStateMachine
GET
UnifiedProgramStateMachine := ADR(_StateMachine);
END_GET
END_PROPERTY

END_FUNCTION_BLOCK

// ---- StateMachine/UnifiedProgram/UnifiedProgramStateMachine.TcPOU
{attribute 'no_explicit_call' := 'do not call this function block directly'}
FUNCTION_BLOCK UnifiedProgramStateMachine EXTENDS ProgramStateMachine
VAR_OUTPUT
	{attribute 'OPC.UA.DA.Access' := '1'}
	Configuration : UNIFIED_PROGRAM_CONFIGURATION;
	
	{attribute 'OPC.UA.DA.Access' := '1'}
	HaltedState : HaltedUnifiedProgramState;
	{attribute 'OPC.UA.DA.Access' := '1'}
	ReadyState : ReadyUnifiedProgramState;
	{attribute 'OPC.UA.DA.Access' := '1'}
	RunningState : RunningUnifiedProgramState;
	{attribute 'OPC.UA.DA.Access' := '1'}
	SuspendedState : SuspendedUnifiedProgramState;
	
	{attribute 'OPC.UA.DA.Access' := '1'}
	HaltedToReady : HaltedToReadyUnifiedProgramTransition;
	{attribute 'OPC.UA.DA.Access' := '1'}
	ReadyToRunning : ReadyToRunningUnifiedProgramTransition;
	{attribute 'OPC.UA.DA.Access' := '1'}
	RunningToHalted : RunningToHaltedUnifiedProgramTransition;
	{attribute 'OPC.UA.DA.Access' := '1'}
	RunningToReady : RunningToReadyUnifiedProgramTransition;
	{attribute 'OPC.UA.DA.Access' := '1'}
	RunningToSuspended : RunningToSuspendedUnifiedProgramTransition;
	{attribute 'OPC.UA.DA.Access' := '1'}
	SuspendedToRunning : SuspendedToRunningUnifiedProgramTransition;
	{attribute 'OPC.UA.DA.Access' := '1'}
	SuspendedToHalted : SuspendedToHaltedUnifiedProgramTransition;
	{attribute 'OPC.UA.DA.Access' := '1'}
	SuspendedToReady : SuspendedToReadyUnifiedProgramTransition;
	{attribute 'OPC.UA.DA.Access' := '1'}
	ReadyToHalted : ReadyToHaltedUnifiedProgramTransition;
	
	{attribute 'OPC.UA.DA' := '0'}
	StepExecutor : UnifiedProgramStepExecutor(THIS^);
END_VAR
VAR_STAT
	//! <summary>Class name shared by all instances of this function block.</summary>
	{attribute 'OPC.UA.DA' := '0'}
	_ClassName : STRING := __POUNAME();
END_VAR

{attribute 'monitoring' := 'call'}
PROPERTY ClassName : REFERENCE TO STRING
GET
ClassName REF= _ClassName;
END_GET
END_PROPERTY

METHOD FB_init : BOOL
VAR_INPUT
	bInitRetains : BOOL; // TRUE: the retain variables are initialized (reset warm / reset cold)
	bInCopyCode : BOOL;  // TRUE: the instance will be copied to the copy code afterward (online change)
END_VAR
JsonHelper.SetFormatOptions(10, EJsonPrettyFormatOptions.eFormatSingleLineArray, 9, 1);
END_METHOD

{attribute 'TcRpcEnable':='1'}
METHOD GetConfiguration : JSON_DOCUMENT
JsonHelper.CreateJsonFromStructure(ADR(Configuration), SIZEOF(Configuration), GetConfiguration);
END_METHOD

METHOD PROTECTED GetStateAndTransitionInstances
VAR_OUTPUT
	haltedState : POINTER TO HaltedProgramState;
	readyState : POINTER TO ReadyProgramState;
	runningState : POINTER TO RunningProgramState;
	suspendedState : POINTER TO SuspendedProgramState;
	
	haltedToReady : POINTER TO HaltedToReadyProgramTransition;
	readyToRunning : POINTER TO ReadyToRunningProgramTransition;
	runningToHalted : POINTER TO RunningToHaltedProgramTransition;
	runningToReady : POINTER TO RunningToReadyProgramTransition;
	runningToSuspended : POINTER TO RunningToSuspendedProgramTransition;
	suspendedToRunning : POINTER TO SuspendedToRunningProgramTransition;
	suspendedToHalted : POINTER TO SuspendedToHaltedProgramTransition;
	suspendedToReady : POINTER TO SuspendedToReadyProgramTransition;
	readyToHalted : POINTER TO ReadyToHaltedProgramTransition;	
END_VAR
haltedState := ADR(THIS^.HaltedState);
readyState := ADR(THIS^.ReadyState);
runningState := ADR(THIS^.RunningState);
suspendedState := ADR(THIS^.SuspendedState);

haltedToReady := ADR(THIS^.HaltedToReady);
readyToRunning := ADR(THIS^.ReadyToRunning);
runningToHalted := ADR(THIS^.RunningToHalted);
runningToReady := ADR(THIS^.RunningToReady);
runningToSuspended := ADR(THIS^.RunningToSuspended);
suspendedToRunning := ADR(THIS^.SuspendedToRunning);
suspendedToHalted := ADR(THIS^.SuspendedToHalted);
suspendedToReady := ADR(THIS^.SuspendedToReady);
readyToHalted := ADR(THIS^.ReadyToHalted);
END_METHOD

METHOD PROTECTED InternalInitialize 
VAR_OUTPUT
	states : ARRAY [0..ProgramConstants.MaxStateCount - 1] OF POINTER TO ProgramState;
	transitions : ARRAY [0..ProgramConstants.MaxTransitionCount - 1] OF POINTER TO ProgramTransition;
	defaultState : POINTER TO ProgramState;
END_VAR
VAR
	haltedState : POINTER TO HaltedProgramState;
	readyState : POINTER TO ReadyProgramState;
	runningState : POINTER TO RunningProgramState;
	suspendedState : POINTER TO SuspendedProgramState;
	
	haltedToReady : POINTER TO HaltedToReadyProgramTransition;
	readyToRunning : POINTER TO ReadyToRunningProgramTransition;
	runningToHalted : POINTER TO RunningToHaltedProgramTransition;
	runningToReady : POINTER TO RunningToReadyProgramTransition;
	runningToSuspended : POINTER TO RunningToSuspendedProgramTransition;
	suspendedToRunning : POINTER TO SuspendedToRunningProgramTransition;
	suspendedToHalted : POINTER TO SuspendedToHaltedProgramTransition;
	suspendedToReady : POINTER TO SuspendedToReadyProgramTransition;
	readyToHalted : POINTER TO ReadyToHaltedProgramTransition;	
END_VAR
END_METHOD

{attribute 'TcRpcEnable':='1'}
METHOD SetConfiguration
VAR_INPUT
	json : JSON_DOCUMENT;
END_VAR
JsonHelper.SetStructureFromJson(json, ADR(Configuration), SIZEOF(Configuration));
END_METHOD

END_FUNCTION_BLOCK

// ---- StateMachine/UnifiedProgram/Transitions/RunningToHaltedUnifiedProgramTransition.TcPOU
FUNCTION_BLOCK RunningToHaltedUnifiedProgramTransition EXTENDS RunningToHaltedProgramTransition
VAR_STAT
	//! <summary>Class name shared by all instances of this function block.</summary>
	{attribute 'OPC.UA.DA' := '0'}
	_ClassName : STRING := __POUNAME();
END_VAR

{attribute 'monitoring' := 'call'}
PROPERTY ClassName : REFERENCE TO STRING
GET
ClassName REF= _ClassName;
END_GET
END_PROPERTY

END_FUNCTION_BLOCK

// ---- StateMachine/UnifiedProgram/Transitions/RunningToReadyUnifiedProgramTransition.TcPOU
FUNCTION_BLOCK RunningToReadyUnifiedProgramTransition EXTENDS RunningToReadyProgramTransition
VAR_STAT
	//! <summary>Class name shared by all instances of this function block.</summary>
	{attribute 'OPC.UA.DA' := '0'}
	_ClassName : STRING := __POUNAME();
END_VAR

{attribute 'monitoring' := 'call'}
PROPERTY ClassName : REFERENCE TO STRING
GET
ClassName REF= _ClassName;
END_GET
END_PROPERTY

END_FUNCTION_BLOCK

// ---- StateMachine/UnifiedProgram/Transitions/RunningToSuspendedUnifiedProgramTransition.TcPOU
FUNCTION_BLOCK RunningToSuspendedUnifiedProgramTransition EXTENDS RunningToSuspendedProgramTransition
VAR_STAT
	//! <summary>Class name shared by all instances of this function block.</summary>
	{attribute 'OPC.UA.DA' := '0'}
	_ClassName : STRING := __POUNAME();
END_VAR

{attribute 'monitoring' := 'call'}
PROPERTY ClassName : REFERENCE TO STRING
GET
ClassName REF= _ClassName;
END_GET
END_PROPERTY

END_FUNCTION_BLOCK

// ---- StateMachine/UnifiedProgram/Transitions/SuspendedToRunningUnifiedProgramTransition.TcPOU
FUNCTION_BLOCK SuspendedToRunningUnifiedProgramTransition EXTENDS SuspendedToRunningProgramTransition
VAR_STAT
	//! <summary>Class name shared by all instances of this function block.</summary>
	{attribute 'OPC.UA.DA' := '0'}
	_ClassName : STRING := __POUNAME();
END_VAR

{attribute 'monitoring' := 'call'}
PROPERTY ClassName : REFERENCE TO STRING
GET
ClassName REF= _ClassName;
END_GET
END_PROPERTY

END_FUNCTION_BLOCK

// ---- StateMachine/UnifiedProgram/Transitions/SuspendedToHaltedUnifiedProgramTransition.TcPOU
FUNCTION_BLOCK SuspendedToHaltedUnifiedProgramTransition EXTENDS SuspendedToHaltedProgramTransition
VAR_STAT
	//! <summary>Class name shared by all instances of this function block.</summary>
	{attribute 'OPC.UA.DA' := '0'}
	_ClassName : STRING := __POUNAME();
END_VAR

{attribute 'monitoring' := 'call'}
PROPERTY ClassName : REFERENCE TO STRING
GET
ClassName REF= _ClassName;
END_GET
END_PROPERTY

END_FUNCTION_BLOCK

// ---- StateMachine/UnifiedProgram/Transitions/SuspendedToReadyUnifiedProgramTransition.TcPOU
FUNCTION_BLOCK SuspendedToReadyUnifiedProgramTransition EXTENDS SuspendedToReadyProgramTransition
VAR_STAT
	//! <summary>Class name shared by all instances of this function block.</summary>
	{attribute 'OPC.UA.DA' := '0'}
	_ClassName : STRING := __POUNAME();
END_VAR

{attribute 'monitoring' := 'call'}
PROPERTY ClassName : REFERENCE TO STRING
GET
ClassName REF= _ClassName;
END_GET
END_PROPERTY

END_FUNCTION_BLOCK

// ---- StateMachine/UnifiedProgram/UnifiedProgramStepExecutor.TcPOU
{attribute 'no_explicit_call' := 'do not call this function block directly'}
{attribute 'OPC.UA.DA' := '0'}
FUNCTION_BLOCK INTERNAL UnifiedProgramStepExecutor EXTENDS ToolkitObject
VAR_STAT
	//! <summary>Class name shared by all instances of this function block.</summary>
	_ClassName : STRING := __POUNAME();
END_VAR
VAR
	_StateMachine : REFERENCE TO UnifiedProgramStateMachine;
	
	_ExecutedSteps : ARRAY [0..UnifiedProgramConstants.MaxStepCount - 1] OF UNIFIED_PROGRAM_EXECUTED_STEP;
	_ExecutedStepCount : INT;
	_ExecutedStep : REFERENCE TO UNIFIED_PROGRAM_EXECUTED_STEP;	
END_VAR

{attribute 'monitoring' := 'call'}
PROPERTY ClassName : REFERENCE TO STRING
GET
ClassName REF= _ClassName;
END_GET
END_PROPERTY

METHOD FB_init : BOOL
VAR_INPUT
	bInitRetains : BOOL; // TRUE: the retain variables are initialized (reset warm / reset cold)
	bInCopyCode : BOOL;  // TRUE: the instance will be copied to the copy code afterward (online change)
	stateMachine : REFERENCE TO UnifiedProgramStateMachine;
END_VAR
_StateMachine REF= stateMachine;
END_METHOD

METHOD Reset 
VAR
	i : DINT;
END_VAR
FOR i := 0 TO UnifiedProgramConstants.MaxStepCount - 1 DO
	_ExecutedSteps[i].StepIndex := -1;
	_ExecutedSteps[i].Step REF= 0;
END_FOR

_ExecutedStepCount := 0;
_ExecutedStep REF= 0;
END_METHOD

END_FUNCTION_BLOCK
